// TIA Portal project "Auto_Gate" (V17)
// This proget is to carry  a simulation of the funtiong on of automatic gates, thsi project should allow us test the consept of position controled feedback systems

(* hardware
DEVICE "S7-300/ET200M station_1"  S7-300 station
   slot 0: "Rail_0"  Rail  6ES7 390-1***0-0AA0
   slot 2: "PLC_1"  CPU 314C-2 PN/DP  6ES7 314-6EH04-0AB0  V3.3
      slot 2: "PROFINET interface_1"  PN-IO
         slot 1: "Port_1"  Port
         slot 2: "Port_2"  Port
      slot 5: "DI 24/DO 16_1"  DI24/DO16
      slot 6: "AI 5/AO 2_1"  AI5/AO2
      slot 7: "Count_1"  Counter
      slot 8: "Positioning_1"  Positioning
*)

// ===== PLC "PLC_1"  CPU 314C-2 PN/DP =====

VAR_GLOBAL   // PLC tag table "Default tag table"
   "Q0.2" AT %Q0.2 : Bool;
   "Q0.0" AT %Q0.0 : Bool;
   "I0.0" AT %I0.0 : Bool;
   "I0.3" AT %I0.3 : Bool;
   "I0.1" AT %I0.1 : Bool;
   "I0.2" AT %I0.2 : Bool;
   "Q0.1" AT %Q0.1 : Bool;
   "Q0.3" AT %Q0.3 : Bool;
   "I0.4" AT %I0.4 : Bool;
END_VAR

TYPE "Auto_Gate"
   STRUCT
      "I0.0" : Bool;
      "I0.1" : Bool;
      "I0.2" : Bool;
      "I0.3" : Bool;
      "I0.4" : Bool;
      "Q0.0" : Bool;
      "Q0.1" : Bool;
      "Q0.2" : Bool;
      "Q0.3" : Bool;
   END_STRUCT;
END_TYPE

ORGANIZATION_BLOCK "Auto_Gate_m"   // OB1, LAD
TITLE = "Main Program Sweep (Cycle)"
{ S7_Optimized_Access := 'FALSE' }
VERSION : 0.1
   VAR_TEMP
      OB1_EV_CLASS : Byte;   // Bits 0-3 = 1 (Coming event), Bits 4-7 = 1 (Event class 1)
      OB1_SCAN_1 : Byte;   // 1 (Cold restart scan 1 of OB 1), 3 (Scan 2-n of OB 1)
      OB1_PRIORITY : Byte;   // Priority of OB Execution
      OB1_OB_NUMBR : Byte;   // 1 (Organization block 1, OB1)
      OB1_RESERVED_1 : Byte;   // Reserved for system
      OB1_RESERVED_2 : Byte;   // Reserved for system
      OB1_PREV_CYCLE : Int;   // Cycle time of previous OB1 scan (milliseconds)
      OB1_MIN_CYCLE : Int;   // Minimum cycle time of OB1 (milliseconds)
      OB1_MAX_CYCLE : Int;   // Maximum cycle time of OB1 (milliseconds)
      OB1_DATE_TIME : Date_And_Time;   // Date and time OB1 started
   END_VAR
BEGIN

REGION Network 1
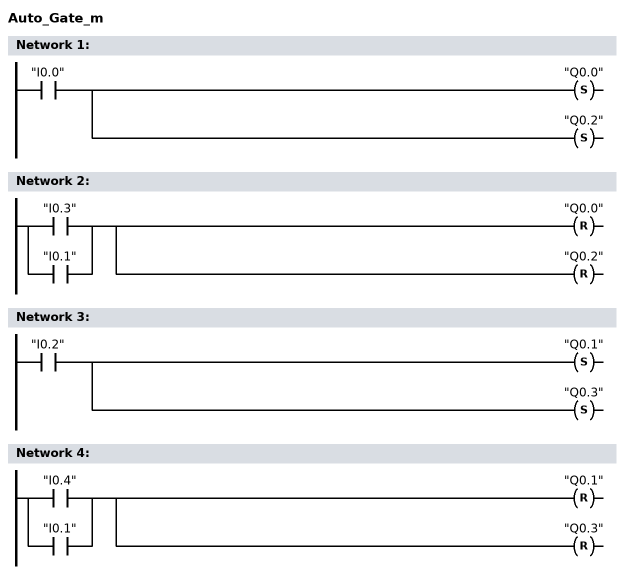
   RUNG wire#powerrail
      Contact( "I0.0" )
      wire#w1
      S_Coil( "Q0.0" )
   END_RUNG
   RUNG wire#w1
      S_Coil( "Q0.2" )
   END_RUNG
   // the same network as SCL:
   IF "I0.0" THEN
       "Q0.0" := TRUE;
       "Q0.2" := TRUE;
   END_IF;
END_REGION

REGION Network 2
   RUNG wire#powerrail
      Contact( "I0.3" )
      wire#w1
      R_Coil( "Q0.0" )
   END_RUNG
   RUNG wire#powerrail
      Contact( "I0.1" )
   END_RUNG wire#w1
   RUNG wire#w1
      R_Coil( "Q0.2" )
   END_RUNG
   // the same network as SCL:
   IF "I0.3" OR "I0.1" THEN
       "Q0.0" := FALSE;
       "Q0.2" := FALSE;
   END_IF;
END_REGION

REGION Network 3
   RUNG wire#powerrail
      Contact( "I0.2" )
      wire#w1
      S_Coil( "Q0.1" )
   END_RUNG
   RUNG wire#w1
      S_Coil( "Q0.3" )
   END_RUNG
   // the same network as SCL:
   IF "I0.2" THEN
       "Q0.1" := TRUE;
       "Q0.3" := TRUE;
   END_IF;
END_REGION

REGION Network 4
   RUNG wire#powerrail
      Contact( "I0.4" )
      wire#w1
      R_Coil( "Q0.1" )
   END_RUNG
   RUNG wire#powerrail
      Contact( "I0.1" )
   END_RUNG wire#w1
   RUNG wire#w1
      R_Coil( "Q0.3" )
   END_RUNG
   // the same network as SCL:
   IF "I0.4" OR "I0.1" THEN
       "Q0.1" := FALSE;
       "Q0.3" := FALSE;
   END_IF;
END_REGION
END_ORGANIZATION_BLOCK